TYPE ST_HomeAdsGroup :
STRUCT
    nCalibrationVel			:UDINT:=16#4001;				(* 回零速度ADS地址*)	
	nHomeInfo				:UDINT:=16#5001;				(* 回零参数ADS地址*)

END_STRUCT
END_TYPE

(* stored: Version 1.1.0.1, ProductVersion 3.1.4024.12
   DUT ST_HomeAdsGroup: Id {75bc2609-c953-4dc3-82d2-c6bcc524bae2} *)
